// TIA Portal V20 export
DATA_BLOCK "InstCallEquipment"   // DB130
{ DB_Accessible_From_OPC_UA := 'FALSE' }
AUTHOR : ERsystem_FA2_DH. Kim
// stored: AssignedProDiagFB Unit1.Em6.ProDiag, DBAccessibleFromOPCUA false, DBAccessibleFromWebserver false, InstanceOfName Unit1.Em6.CallEquipment, InstanceOfType FB, Namespace Unit1.Em6
"Unit1.Em6.CallEquipment"
   // VAR_INPUT
   //    ZoneOperationEnable { ExternalWritable := 'False'} : "LWONIK_typeSafetyZoneManualOperation";
   // END_VAR
   // VAR_IN_OUT
   //    unitStatus : "LAF_typeUnitStatus";
   //    unitAlarmDB : "LAF_typeAlarms";
   //    emFeedback : "LUC_typeEmFeedback";
   // END_VAR
   // VAR
   //    InstSequenceStackTable { S7_SetPoint := 'True'} : "Unit1.Em6.Sequence_1_StackTable";
   //    InstSequenceGaugeRnR { S7_SetPoint := 'True'} : "Unit1.Em6.Sequence_10_GaugeRnR";
   //    InstSequenceUtility { S7_SetPoint := 'True'} : "Unit1.Em6.Sequence_20_Utility";
   //    instStackTableHomeJob1 { S7_SetPoint := 'True'} : "LAF_SelectJob";
   //    instStackTableMotionAutoJob2 { S7_SetPoint := 'True'} : "LAF_SelectJob";
   //    instStackTableRollerMoveJob12 { S7_SetPoint := 'True'} : "LAF_SelectJob";
   //    instStackTableRollerMoveJob13 { S7_SetPoint := 'True'} : "LAF_SelectJob";
   //    instStackTableSepaCleanJob14 { S7_SetPoint := 'True'} : "LAF_SelectJob";
   //    instStackTableAnodeMendrelJob22 { S7_SetPoint := 'True'} : "LAF_SelectJob";
   //    instStackTableCathodeMendrelJob23 { S7_SetPoint := 'True'} : "LAF_SelectJob";
   //    instStackTableVisionJob30 { S7_SetPoint := 'True'} : "LAF_SelectJob";
   //    instStackTableDownJob31 { S7_SetPoint := 'True'} : "LAF_SelectJob";
   //    instStackTableUnloadJob4 { S7_SetPoint := 'True'} : "LAF_SelectJob";
   //    instGaugeRnRReadyJob1 { S7_SetPoint := 'True'} : "LAF_SelectJob";
   //    instGaugeRnRVaccumJob2 { S7_SetPoint := 'True'} : "LAF_SelectJob";
   //    instGaugeRnRVisionJob3 { S7_SetPoint := 'True'} : "LAF_SelectJob";
   //    instGaugeRnRBlowJob4 { S7_SetPoint := 'True'} : "LAF_SelectJob";
   //    instUtilityFinalRollerHomeJob1 { S7_SetPoint := 'True'} : "LAF_SelectJob";
   //    instUtilityStackTableOutHomeJob2 { S7_SetPoint := 'True'} : "LAF_SelectJob";
   //    instUtilityAllMendrelOpenJob3 { S7_SetPoint := 'True'} : "LAF_SelectJob";
   //    instUtilityAllMendrelCloseJob4 { S7_SetPoint := 'True'} : "LAF_SelectJob";
   //    instCmStackTableElectrodeDetectSensor { S7_SetPoint := 'True'} : "LBC_DigitalSignalCn";
   //    instCmMasterVirtualAxisX : "LBC_Axis64Pos_TecPlcCn";
   //    instCmFinalRollerFrontAxisX : "LBC_Axis64Pos_TecPlcCn";
   //    instCmFinalRollerRearAxisX { S7_SetPoint := 'True'} : "LBC_Axis64Pos_TecPlcCn";
   //    instCmMendrelAnodeFrontAxisY { S7_SetPoint := 'True'} : "LBC_Axis64Pos_TecPlcCn";
   //    instCmMendrelAnodeFrontAxisZ { S7_SetPoint := 'True'} : "LBC_Axis64Pos_TecPlcCn";
   //    instCmMendrelAnodeRearAxisY { S7_SetPoint := 'True'} : "LBC_Axis64Pos_TecPlcCn";
   //    instCmMendrelAnodeRearAxisZ { S7_SetPoint := 'True'} : "LBC_Axis64Pos_TecPlcCn";
   //    instCmMendrelCathodeFrontAxisY { S7_SetPoint := 'True'} : "LBC_Axis64Pos_TecPlcCn";
   //    instCmMendrelCathodeFrontAxisZ { S7_SetPoint := 'True'} : "LBC_Axis64Pos_TecPlcCn";
   //    instCmMendrelCathodeRearAxisY { S7_SetPoint := 'True'} : "LBC_Axis64Pos_TecPlcCn";
   //    instCmMendrelCathodeRearAxisZ { S7_SetPoint := 'True'} : "LBC_Axis64Pos_TecPlcCn";
   //    instCmStackTableAxisZ { ExternalAccessible := 'False'; ExternalVisible := 'False'; ExternalWritable := 'False'; S7_SetPoint := 'True'} : "LBC_Axis64Pos_TecPlcCn";
   //    instCmStackTableOutFrontAxisZ { ExternalAccessible := 'False'; ExternalVisible := 'False'; ExternalWritable := 'False'; S7_SetPoint := 'True'} : "LBC_Axis64Pos_TecPlcCn";
   //    instCmStackTableOutRearAxisZ { ExternalAccessible := 'False'; ExternalVisible := 'False'; ExternalWritable := 'False'; S7_SetPoint := 'True'} : "LBC_Axis64Pos_TecPlcCn";
   //    instInterlockFinalRollerFrontAxisX : "LER_Axis64Pos_InterlockSummary";
   //    instInterlockFinalRollerRearAxisX : "LER_Axis64Pos_InterlockSummary";
   //    instInterlockMendrelAnodeFrontAxisY : "LER_Axis64Pos_InterlockSummary";
   //    instInterlockMendrelAnodeFrontAxisZ : "LER_Axis64Pos_InterlockSummary";
   //    instInterlockMendrelAnodeRearAxisY : "LER_Axis64Pos_InterlockSummary";
   //    instInterlockMendrelAnodeRearAxisZ : "LER_Axis64Pos_InterlockSummary";
   //    instInterlockMendrelCathodeFrontAxisY : "LER_Axis64Pos_InterlockSummary";
   //    instInterlockMendrelCathodeFrontAxisZ : "LER_Axis64Pos_InterlockSummary";
   //    instInterlockMendrelCathodeRearAxisY : "LER_Axis64Pos_InterlockSummary";
   //    instInterlockMendrelCathodeRearAxisZ : "LER_Axis64Pos_InterlockSummary";
   //    instInterlockStackTableAxisZ : "LER_Axis64Pos_InterlockSummary";
   //    instInterlockStackTableOutFrontAxisZ : "LER_Axis64Pos_InterlockSummary";
   //    instInterlockStackTableOutRearAxisZ : "LER_Axis64Pos_InterlockSummary";
   //    instFinalRollerFrontAxisXMCGearIn { S7_SetPoint := 'True'} : MC_GEARIN;
   //    instFinalRollerRearAxisXMCGearIn { S7_SetPoint := 'True'} : MC_GEARIN;
   //    instStackTableOutFrontAxisZMCGearIn { S7_SetPoint := 'True'} : MC_GEARIN;
   //    instStackTableOutRearAxisZMCGearIn { S7_SetPoint := 'True'} : MC_GEARIN;
   //    instFinalRollerFrontAxisXMCWirteParameter { S7_SetPoint := 'True'} : MC_WRITEPARAMETER;
   //    instFinalRollerRearAxisXMCWirteParameter { S7_SetPoint := 'True'} : MC_WRITEPARAMETER;
   //    instStackTableOutFrontAxisZMCWirteParameter { S7_SetPoint := 'True'} : MC_WRITEPARAMETER;
   //    instStackTableOutRearAxisZMCWirteParameter { S7_SetPoint := 'True'} : MC_WRITEPARAMETER;
   //    instCmMendrelCathodeFrontClamp { ExternalAccessible := 'False'; ExternalVisible := 'False'; ExternalWritable := 'False'; S7_SetPoint := 'True'} : "LBC_TwoWayActuatorCn";
   //    instCmMendrelAnodeFrontClamp { ExternalAccessible := 'False'; ExternalVisible := 'False'; ExternalWritable := 'False'; S7_SetPoint := 'True'} : "LBC_TwoWayActuatorCn";
   //    instCmMendrelCathodeRearClamp { ExternalAccessible := 'False'; ExternalVisible := 'False'; ExternalWritable := 'False'; S7_SetPoint := 'True'} : "LBC_TwoWayActuatorCn";
   //    instCmMendrelAnodeRearClamp { ExternalAccessible := 'False'; ExternalVisible := 'False'; ExternalWritable := 'False'; S7_SetPoint := 'True'} : "LBC_TwoWayActuatorCn";
   //    instcmStackTableVaccum { ExternalAccessible := 'False'; ExternalVisible := 'False'; ExternalWritable := 'False'; S7_SetPoint := 'True'} : "LBC_TwoWayActuatorCn";
   //    instcmStackTableGapPadUpDown { ExternalAccessible := 'False'; ExternalVisible := 'False'; ExternalWritable := 'False'; S7_SetPoint := 'True'} : "LBC_TwoWayActuatorCn";
   //    instCmStackTableVisionControllerInterface : "LER_Vision_XGX2000";
   //    instGapVisionConversion : "LER_StackTableVisionConversion";
   //    instManageAlarms { ExternalWritable := 'False'} : "LAF_ManageAlarms";
   //    instEventsPFE : "Unit1.Em6.EventsPFE";
   //    instLER_BrakeTestMendrelAnodeFrontAxisZ : "LER_BrakeTest";
   //    instLER_BrakeTestMendrelAnodeRearAxisZ { S7_SetPoint := 'True'} : "LER_BrakeTest";
   //    instLER_BrakeTestMendrelCathodeFrontAxisZ { S7_SetPoint := 'True'} : "LER_BrakeTest";
   //    instLER_BrakeTestMendrelCathodeRearAxisZ { S7_SetPoint := 'True'} : "LER_BrakeTest";
   //    instLER_BrakeTestStackTableAxisZ { S7_SetPoint := 'True'} : "LER_BrakeTest";
   //    instLER_BrakeTestStackTableOutFrontAxisZ { S7_SetPoint := 'True'} : "LER_BrakeTest";
   //    instLER_BrakeTestStackTableOutRearAxisZ { S7_SetPoint := 'True'} : "LER_BrakeTest";
   //    statUnitStatus { ExternalWritable := 'False'} : "LAF_typeUnitStatus";
   //    statSlmStatus : Struct
   //       running { ExternalWritable := 'False'} : Bool;
   //       powerOff { ExternalWritable := 'False'} : Bool;
   //    END_STRUCT;
   //    statAllBrakeTest { ExternalWritable := 'False'} : "LER_typeBrakeTestUnitCommands";
   //    statTonTime { ExternalAccessible := 'False'; ExternalVisible := 'False'; ExternalWritable := 'False'} : Array[0..1999] of TON_TIME;
   //    statTofTime { ExternalAccessible := 'False'; ExternalVisible := 'False'; ExternalWritable := 'False'} : Array[0..99] of TOF_TIME;
   //    statLReal { ExternalAccessible := 'False'; ExternalVisible := 'False'; ExternalWritable := 'False'} : Array[0..99] of LReal;
   //    statPulse { ExternalAccessible := 'False'; ExternalVisible := 'False'; ExternalWritable := 'False'} : Struct
   //       miscellaneous : Array[0..99] of Bool;
   //       workingDone : Array[0..99] of Bool;
   //       axisEnable : Array[0..99] of Bool;
   //       brakeTest : Array[0..99] of Bool;
   //    END_STRUCT;
   //    statEnableManualCmds : Bool := TRUE;
   //    scan_on : Bool;
   //    "*** Interlock Axis ***" { ExternalAccessible := 'False'; ExternalVisible := 'False'; ExternalWritable := 'False'} : Bool;
   //    instFinalRollerFrontAxisX_CW { S7_SetPoint := 'True'} : "Jog.LER_Axis";
   //    instFinalRollerFrontAxisX_CCW { S7_SetPoint := 'True'} : "Jog.LER_Axis";
   //    instFinalRollerFrontAxisX_Home { S7_SetPoint := 'True'} : "Homing.LER_Axis";
   //    instFinalRollerFrontAxisX_Position { S7_SetPoint := 'True'} : Array[0..6] of "Position.LER_Axis";
   //    instFinalRollerRearAxisX_CW { S7_SetPoint := 'True'} : "Jog.LER_Axis";
   //    instFinalRollerRearAxisX_CCW { S7_SetPoint := 'True'} : "Jog.LER_Axis";
   //    instFinalRollerRearAxisX_Home { S7_SetPoint := 'True'} : "Homing.LER_Axis";
   //    instFinalRollerRearAxisX_Position { S7_SetPoint := 'True'} : Array[0..6] of "Position.LER_Axis";
   //    instMendrelAnodeFrontAxisY_CW { S7_SetPoint := 'True'} : "Jog.LER_Axis";
   //    instMendrelAnodeFrontAxisY_CCW { S7_SetPoint := 'True'} : "Jog.LER_Axis";
   //    instMendrelAnodeFrontAxisY_Home { S7_SetPoint := 'True'} : "Homing.LER_Axis";
   //    instMendrelAnodeFrontAxisY_Position { S7_SetPoint := 'True'} : Array[0..15] of "Position.LER_Axis";
   //    instMendrelAnodeFrontAxisZ_CW { S7_SetPoint := 'True'} : "Jog.LER_Axis";
   //    instMendrelAnodeFrontAxisZ_CCW { S7_SetPoint := 'True'} : "Jog.LER_Axis";
   //    instMendrelAnodeFrontAxisZ_Home { S7_SetPoint := 'True'} : "Homing.LER_Axis";
   //    instMendrelAnodeFrontAxisZ_Position { S7_SetPoint := 'True'} : Array[0..6] of "Position.LER_Axis";
   //    instMendrelAnodeRearAxisY_CW { S7_SetPoint := 'True'} : "Jog.LER_Axis";
   //    instMendrelAnodeRearAxisY_CCW { S7_SetPoint := 'True'} : "Jog.LER_Axis";
   //    instMendrelAnodeRearAxisY_Home { S7_SetPoint := 'True'} : "Homing.LER_Axis";
   //    instMendrelAnodeRearAxisY_Position { S7_SetPoint := 'True'} : Array[0..6] of "Position.LER_Axis";
   //    instMendrelAnodeRearAxisZ_CW { S7_SetPoint := 'True'} : "Jog.LER_Axis";
   //    instMendrelAnodeRearAxisZ_CCW { S7_SetPoint := 'True'} : "Jog.LER_Axis";
   //    instMendrelAnodeRearAxisZ_Home { S7_SetPoint := 'True'} : "Homing.LER_Axis";
   //    instMendrelAnodeRearAxisZ_Position { S7_SetPoint := 'True'} : Array[0..6] of "Position.LER_Axis";
   //    instMendrelCathodeFrontAxisY_CW { S7_SetPoint := 'True'} : "Jog.LER_Axis";
   //    instMendrelCathodeFrontAxisY_CCW { S7_SetPoint := 'True'} : "Jog.LER_Axis";
   //    instMendrelCathodeFrontAxisY_Home { S7_SetPoint := 'True'} : "Homing.LER_Axis";
   //    instMendrelCathodeFrontAxisY_Position { S7_SetPoint := 'True'} : Array[0..6] of "Position.LER_Axis";
   //    instMendrelCathodeFrontAxisZ_CW { S7_SetPoint := 'True'} : "Jog.LER_Axis";
   //    instMendrelCathodeFrontAxisZ_CCW { S7_SetPoint := 'True'} : "Jog.LER_Axis";
   //    instMendrelCathodeFrontAxisZ_Home { S7_SetPoint := 'True'} : "Homing.LER_Axis";
   //    instMendrelCathodeFrontAxisZ_Position { S7_SetPoint := 'True'} : Array[0..6] of "Position.LER_Axis";
   //    instMendrelCathodeRearAxisY_CW { S7_SetPoint := 'True'} : "Jog.LER_Axis";
   //    instMendrelCathodeRearAxisY_CCW { S7_SetPoint := 'True'} : "Jog.LER_Axis";
   //    instMendrelCathodeRearAxisY_Home { S7_SetPoint := 'True'} : "Homing.LER_Axis";
   //    instMendrelCathodeRearAxisY_Position { S7_SetPoint := 'True'} : Array[0..6] of "Position.LER_Axis";
   //    instMendrelCathodeRearAxisZ_CW { S7_SetPoint := 'True'} : "Jog.LER_Axis";
   //    instMendrelCathodeRearAxisZ_CCW { S7_SetPoint := 'True'} : "Jog.LER_Axis";
   //    instMendrelCathodeRearAxisZ_Home { S7_SetPoint := 'True'} : "Homing.LER_Axis";
   //    instMendrelCathodeRearAxisZ_Position { S7_SetPoint := 'True'} : Array[0..6] of "Position.LER_Axis";
   //    instStackTableAxisZ_CW { S7_SetPoint := 'True'} : "Jog.LER_Axis";
   //    instStackTableAxisZ_CCW { S7_SetPoint := 'True'} : "Jog.LER_Axis";
   //    instStackTableAxisZ_Home { S7_SetPoint := 'True'} : "Homing.LER_Axis";
   //    instStackTableAxisZ_Position { S7_SetPoint := 'True'} : Array[0..6] of "Position.LER_Axis";
   //    instStackTableOutFrontAxisZ_CW { S7_SetPoint := 'True'} : "Jog.LER_Axis";
   //    instStackTableOutFrontAxisZ_CCW { S7_SetPoint := 'True'} : "Jog.LER_Axis";
   //    instStackTableOutFrontAxisZ_Home { S7_SetPoint := 'True'} : "Homing.LER_Axis";
   //    instStackTableOutFrontAxisZ_Position { S7_SetPoint := 'True'} : Array[0..6] of "Position.LER_Axis";
   //    instStackTableOutRearAxisZ_CW { S7_SetPoint := 'True'} : "Jog.LER_Axis";
   //    instStackTableOutRearAxisZ_CCW { S7_SetPoint := 'True'} : "Jog.LER_Axis";
   //    instStackTableOutRearAxisZ_Home { S7_SetPoint := 'True'} : "Homing.LER_Axis";
   //    instStackTableOutRearAxisZ_Position { S7_SetPoint := 'True'} : Array[0..6] of "Position.LER_Axis";
   //    "*** Interlock Actuator ******" { ExternalAccessible := 'False'; ExternalVisible := 'False'; ExternalWritable := 'False'} : Bool;
   //    instCmMendrelCathodeFrontClampInterlock : Array[0..1] of "Cylinder.LER_Actuator";
   //    instCmMendrelAnodeFrontClampInterlock { S7_SetPoint := 'True'} : Array[0..1] of "Cylinder.LER_Actuator";
   //    instCmMendrelCathodeRearClampInterlock { S7_SetPoint := 'True'} : Array[0..1] of "Cylinder.LER_Actuator";
   //    instCmMendrelAnodeRearClampInterlock { S7_SetPoint := 'True'} : Array[0..1] of "Cylinder.LER_Actuator";
   //    instcmStackTableVaccumInterlock { S7_SetPoint := 'True'} : Array[0..1] of "Cylinder.LER_Actuator";
   //    instcmStackTableGapPadUpDownInterlock { S7_SetPoint := 'True'} : Array[0..1] of "Cylinder.LER_Actuator";
   //    AXIS21 : "LER_CM_Name";
   //    AXIS26 : "LER_CM_Name";
   //    AXIS31 : "LER_CM_Name";
   //    Cylinder33 : "LER_CM_Name";
   //    Vaccum20 : "LER_CM_Name";
   //    instFinalRollerGearInVel : MC_GEARINVELOCITY;
   //    instStackTableOutGearInVel : MC_GEARINVELOCITY;
   //    instFinalRollerGantryHoming : "LER_GantryHoming";
   //    instStackTableOutGantryHoming : "LER_GantryHoming";
   //    citi_Ptrig : Array[0..20] of Bool;
   //    citiTon : Array[0..20] of TON_TIME;
   //    citi : Time;
   //    citiTest : Array[0..20] of Bool;
   // END_VAR
BEGIN
   ZoneOperationEnable.autoStartEnable := FALSE;
   ZoneOperationEnable.doorLockEnable := TRUE;
   ZoneOperationEnable.doorUnlockEnable := TRUE;
   ZoneOperationEnable.rc_AutoEnable := FALSE;
   ZoneOperationEnable.rc_RollChangeEnable := FALSE;
   ZoneOperationEnable.rc_DoorLockEnable := TRUE;
   ZoneOperationEnable.rc_DoorUnlockEnable := TRUE;
   ZoneOperationEnable.hmiOperationEnable := TRUE;
   ZoneOperationEnable.phmiOperationEnable := FALSE;
   instCmStackTableElectrodeDetectSensor.enable := TRUE;
   instCmStackTableElectrodeDetectSensor.parentReferenceDesignator := WSTRING#'';
   instCmStackTableElectrodeDetectSensor.digitalValue := FALSE;
   instCmStackTableElectrodeDetectSensor.simulatedDigitalValue := FALSE;
   instCmStackTableElectrodeDetectSensor.statProcessValues.enable := TRUE;
   instCmStackTableElectrodeDetectSensor.statProcessValues.referenceDesignator := WSTRING#'DigitalSignal';
   instCmStackTableElectrodeDetectSensor.statProcessValues.simulation := FALSE;
   instCmStackTableElectrodeDetectSensor.statProcessValues.processValue := FALSE;
   instCmStackTableElectrodeDetectSensor.statProcessValues.error := FALSE;
   instCmStackTableElectrodeDetectSensor.statProcessValues.status := 16#0000;
   instCmStackTableElectrodeDetectSensor.statDiagnostics.status := 16#0000;
   instCmStackTableElectrodeDetectSensor.statDiagnostics.subfunctionStatus := 16#0000;
   instCmStackTableElectrodeDetectSensor.statDiagnostics.stateNumber := 0;
   instCmStackTableElectrodeDetectSensor.statEmptyDiagnostics.status := 16#0000;
   instCmStackTableElectrodeDetectSensor.statEmptyDiagnostics.subfunctionStatus := 16#0000;
   instCmStackTableElectrodeDetectSensor.statEmptyDiagnostics.stateNumber := 0;
   instCmStackTableElectrodeDetectSensor.instOnDelay.PT := T#0MS;
   instCmStackTableElectrodeDetectSensor.instOnDelay.IN := FALSE;
   instCmStackTableElectrodeDetectSensor.instOffDelay.PT := T#0MS;
   instCmStackTableElectrodeDetectSensor.instOffDelay.IN := FALSE;
   instCmStackTableElectrodeDetectSensor.statDisableAlarms := FALSE;
   instCmStackTableElectrodeDetectSensor.statErrorState := 16#0000;
   instCmStackTableElectrodeDetectSensor.statFirstCall := FALSE;
   instCmStackTableElectrodeDetectSensor.statResetPrevious := FALSE;
   instCmStackTableElectrodeDetectSensor.statEnablePrevious := TRUE;
   instCmStackTableElectrodeDetectSensor.statProcessValuePrevious := FALSE;
   instCmMendrelCathodeFrontClamp.enable := TRUE;
   instCmMendrelCathodeFrontClamp.parentReferenceDesignator := WSTRING#'';
   instCmMendrelCathodeFrontClamp.feedbackHomePos := FALSE;
   instCmMendrelCathodeFrontClamp.feedbackWorkPos := FALSE;
   instCmMendrelCathodeFrontClamp.enableManualCmds := TRUE;
   instCmMendrelCathodeFrontClamp.interlockWorkPos := TRUE;
   instCmMendrelCathodeFrontClamp.interlockHomePos := TRUE;
   instCmMendrelCathodeFrontClamp.goToHomePos := FALSE;
   instCmMendrelCathodeFrontClamp.goToWorkPos := FALSE;
   instCmMendrelCathodeFrontClamp.statProcessValues.enable := TRUE;
   instCmMendrelCathodeFrontClamp.statProcessValues.referenceDesignator := WSTRING#'MendrelCathodeFrontClamp';
   instCmMendrelCathodeFrontClamp.statProcessValues.commandHomePos := FALSE;
   instCmMendrelCathodeFrontClamp.statProcessValues.commandWorkPos := FALSE;
   instCmMendrelCathodeFrontClamp.statProcessValues.goToHomePos := FALSE;
   instCmMendrelCathodeFrontClamp.statProcessValues.goToWorkPos := FALSE;
   instCmMendrelCathodeFrontClamp.statProcessValues.inHomePos := FALSE;
   instCmMendrelCathodeFrontClamp.statProcessValues.inWorkPos := FALSE;
   instCmMendrelCathodeFrontClamp.statProcessValues.reset := FALSE;
   instCmMendrelCathodeFrontClamp.statProcessValues.enableManualCmds := TRUE;
   instCmMendrelCathodeFrontClamp.statProcessValues.error := FALSE;
   instCmMendrelCathodeFrontClamp.statProcessValues.interlockHomePos := TRUE;
   instCmMendrelCathodeFrontClamp.statProcessValues.interlockWorkPos := TRUE;
   instCmMendrelCathodeFrontClamp.statProcessValues.status := 16#7003;
   instCmMendrelCathodeFrontClamp.statProcessValues.interlockWarningWorkPos := FALSE;
   instCmMendrelCathodeFrontClamp.statProcessValues.interlockWarningHomePos := FALSE;
   instCmMendrelCathodeFrontClamp.statCurrentInputs.commandHomePos := FALSE;
   instCmMendrelCathodeFrontClamp.statCurrentInputs.commandWorkPos := FALSE;
   instCmMendrelCathodeFrontClamp.statCurrentInputs.reset := FALSE;
   instCmMendrelCathodeFrontClamp.statPreviousInputs.commandHomePos := FALSE;
   instCmMendrelCathodeFrontClamp.statPreviousInputs.commandWorkPos := FALSE;
   instCmMendrelCathodeFrontClamp.statPreviousInputs.reset := FALSE;
   instCmMendrelCathodeFrontClamp.statCurrentInterface.commandHomePos := FALSE;
   instCmMendrelCathodeFrontClamp.statCurrentInterface.commandWorkPos := FALSE;
   instCmMendrelCathodeFrontClamp.statCurrentInterface.reset := FALSE;
   instCmMendrelCathodeFrontClamp.statPreviousInterface.commandHomePos := FALSE;
   instCmMendrelCathodeFrontClamp.statPreviousInterface.commandWorkPos := FALSE;
   instCmMendrelCathodeFrontClamp.statPreviousInterface.reset := FALSE;
   instCmMendrelCathodeFrontClamp.statEmptyDiagnostics.status := 16#0000;
   instCmMendrelCathodeFrontClamp.statEmptyDiagnostics.subfunctionStatus := 16#0000;
   instCmMendrelCathodeFrontClamp.statEmptyDiagnostics.stateNumber := 0;
   instCmMendrelCathodeFrontClamp.instTimerReachPos.PT := T#0MS;
   instCmMendrelCathodeFrontClamp.instTimerReachPos.IN := FALSE;
   instCmMendrelCathodeFrontClamp.instTimerLeavePos.PT := T#0MS;
   instCmMendrelCathodeFrontClamp.instTimerLeavePos.IN := FALSE;
   instCmMendrelCathodeFrontClamp.instTimerDiscrepancyCheck.PT := T#0MS;
   instCmMendrelCathodeFrontClamp.instTimerDiscrepancyCheck.IN := FALSE;
   instCmMendrelCathodeFrontClamp.statDisableAlarms := FALSE;
   instCmMendrelCathodeFrontClamp.statDiagnostics.status := 16#7003;
   instCmMendrelCathodeFrontClamp.statDiagnostics.subfunctionStatus := 16#0000;
   instCmMendrelCathodeFrontClamp.statDiagnostics.stateNumber := 0;
   instCmMendrelCathodeFrontClamp.statEnablePrevious := TRUE;
   instCmMendrelCathodeFrontClamp.statFirstCall := FALSE;
   instCmMendrelCathodeFrontClamp.statResetPrevious := FALSE;
   instCmMendrelCathodeFrontClamp.statValid := TRUE;
   instCmMendrelCathodeFrontClamp.statBusy := TRUE;
   instCmMendrelCathodeFrontClamp.statError := FALSE;
   instCmMendrelCathodeFrontClamp.statInterlockWorkOff := FALSE;
   instCmMendrelCathodeFrontClamp.statInterlockHomeOff := FALSE;
   instCmMendrelCathodeFrontClamp.statFbState := 50;
   instCmMendrelCathodeFrontClamp.statFbStatePrevious := 50;
   instCmMendrelCathodeFrontClamp.statErrorUserCleared := FALSE;
   instCmMendrelCathodeFrontClamp.statErrorAutoCleared := FALSE;
   instCmMendrelCathodeFrontClamp.statErrorState := 16#0000;
   instCmMendrelCathodeFrontClamp.statDisablingCompleted := FALSE;
   instCmMendrelCathodeFrontClamp.statFeedbackHomePos := FALSE;
   instCmMendrelCathodeFrontClamp.statFeedbackWorkPos := FALSE;
   instCmMendrelAnodeFrontClamp.enable := TRUE;
   instCmMendrelAnodeFrontClamp.parentReferenceDesignator := WSTRING#'';
   instCmMendrelAnodeFrontClamp.feedbackHomePos := FALSE;
   instCmMendrelAnodeFrontClamp.feedbackWorkPos := FALSE;
   instCmMendrelAnodeFrontClamp.enableManualCmds := TRUE;
   instCmMendrelAnodeFrontClamp.interlockWorkPos := TRUE;
   instCmMendrelAnodeFrontClamp.interlockHomePos := TRUE;
   instCmMendrelAnodeFrontClamp.goToHomePos := FALSE;
   instCmMendrelAnodeFrontClamp.goToWorkPos := FALSE;
   instCmMendrelAnodeFrontClamp.statProcessValues.enable := TRUE;
   instCmMendrelAnodeFrontClamp.statProcessValues.referenceDesignator := WSTRING#'MendrelAnodeFrontClamp';
   instCmMendrelAnodeFrontClamp.statProcessValues.commandHomePos := FALSE;
   instCmMendrelAnodeFrontClamp.statProcessValues.commandWorkPos := FALSE;
   instCmMendrelAnodeFrontClamp.statProcessValues.goToHomePos := FALSE;
   instCmMendrelAnodeFrontClamp.statProcessValues.goToWorkPos := FALSE;
   instCmMendrelAnodeFrontClamp.statProcessValues.inHomePos := FALSE;
   instCmMendrelAnodeFrontClamp.statProcessValues.inWorkPos := FALSE;
   instCmMendrelAnodeFrontClamp.statProcessValues.reset := FALSE;
   instCmMendrelAnodeFrontClamp.statProcessValues.enableManualCmds := TRUE;
   instCmMendrelAnodeFrontClamp.statProcessValues.error := FALSE;
   instCmMendrelAnodeFrontClamp.statProcessValues.interlockHomePos := TRUE;
   instCmMendrelAnodeFrontClamp.statProcessValues.interlockWorkPos := TRUE;
   instCmMendrelAnodeFrontClamp.statProcessValues.status := 16#7003;
   instCmMendrelAnodeFrontClamp.statProcessValues.interlockWarningWorkPos := FALSE;
   instCmMendrelAnodeFrontClamp.statProcessValues.interlockWarningHomePos := FALSE;
   instCmMendrelAnodeFrontClamp.statCurrentInputs.commandHomePos := FALSE;
   instCmMendrelAnodeFrontClamp.statCurrentInputs.commandWorkPos := FALSE;
   instCmMendrelAnodeFrontClamp.statCurrentInputs.reset := FALSE;
   instCmMendrelAnodeFrontClamp.statPreviousInputs.commandHomePos := FALSE;
   instCmMendrelAnodeFrontClamp.statPreviousInputs.commandWorkPos := FALSE;
   instCmMendrelAnodeFrontClamp.statPreviousInputs.reset := FALSE;
   instCmMendrelAnodeFrontClamp.statCurrentInterface.commandHomePos := FALSE;
   instCmMendrelAnodeFrontClamp.statCurrentInterface.commandWorkPos := FALSE;
   instCmMendrelAnodeFrontClamp.statCurrentInterface.reset := FALSE;
   instCmMendrelAnodeFrontClamp.statPreviousInterface.commandHomePos := FALSE;
   instCmMendrelAnodeFrontClamp.statPreviousInterface.commandWorkPos := FALSE;
   instCmMendrelAnodeFrontClamp.statPreviousInterface.reset := FALSE;
   instCmMendrelAnodeFrontClamp.statEmptyDiagnostics.status := 16#0000;
   instCmMendrelAnodeFrontClamp.statEmptyDiagnostics.subfunctionStatus := 16#0000;
   instCmMendrelAnodeFrontClamp.statEmptyDiagnostics.stateNumber := 0;
   instCmMendrelAnodeFrontClamp.instTimerReachPos.PT := T#0MS;
   instCmMendrelAnodeFrontClamp.instTimerReachPos.IN := FALSE;
   instCmMendrelAnodeFrontClamp.instTimerLeavePos.PT := T#0MS;
   instCmMendrelAnodeFrontClamp.instTimerLeavePos.IN := FALSE;
   instCmMendrelAnodeFrontClamp.instTimerDiscrepancyCheck.PT := T#0MS;
   instCmMendrelAnodeFrontClamp.instTimerDiscrepancyCheck.IN := FALSE;
   instCmMendrelAnodeFrontClamp.statDisableAlarms := FALSE;
   instCmMendrelAnodeFrontClamp.statDiagnostics.status := 16#7003;
   instCmMendrelAnodeFrontClamp.statDiagnostics.subfunctionStatus := 16#0000;
   instCmMendrelAnodeFrontClamp.statDiagnostics.stateNumber := 0;
   instCmMendrelAnodeFrontClamp.statEnablePrevious := TRUE;
   instCmMendrelAnodeFrontClamp.statFirstCall := FALSE;
   instCmMendrelAnodeFrontClamp.statResetPrevious := FALSE;
   instCmMendrelAnodeFrontClamp.statValid := TRUE;
   instCmMendrelAnodeFrontClamp.statBusy := TRUE;
   instCmMendrelAnodeFrontClamp.statError := FALSE;
   instCmMendrelAnodeFrontClamp.statInterlockWorkOff := FALSE;
   instCmMendrelAnodeFrontClamp.statInterlockHomeOff := FALSE;
   instCmMendrelAnodeFrontClamp.statFbState := 50;
   instCmMendrelAnodeFrontClamp.statFbStatePrevious := 50;
   instCmMendrelAnodeFrontClamp.statErrorUserCleared := FALSE;
   instCmMendrelAnodeFrontClamp.statErrorAutoCleared := FALSE;
   instCmMendrelAnodeFrontClamp.statErrorState := 16#0000;
   instCmMendrelAnodeFrontClamp.statDisablingCompleted := FALSE;
   instCmMendrelAnodeFrontClamp.statFeedbackHomePos := FALSE;
   instCmMendrelAnodeFrontClamp.statFeedbackWorkPos := FALSE;
   instCmMendrelCathodeRearClamp.enable := TRUE;
   instCmMendrelCathodeRearClamp.parentReferenceDesignator := WSTRING#'';
   instCmMendrelCathodeRearClamp.feedbackHomePos := FALSE;
   instCmMendrelCathodeRearClamp.feedbackWorkPos := FALSE;
   instCmMendrelCathodeRearClamp.enableManualCmds := TRUE;
   instCmMendrelCathodeRearClamp.interlockWorkPos := TRUE;
   instCmMendrelCathodeRearClamp.interlockHomePos := TRUE;
   instCmMendrelCathodeRearClamp.goToHomePos := FALSE;
   instCmMendrelCathodeRearClamp.goToWorkPos := FALSE;
   instCmMendrelCathodeRearClamp.statProcessValues.enable := TRUE;
   instCmMendrelCathodeRearClamp.statProcessValues.referenceDesignator := WSTRING#'MendrelCathodeRearClamp';
   instCmMendrelCathodeRearClamp.statProcessValues.commandHomePos := FALSE;
   instCmMendrelCathodeRearClamp.statProcessValues.commandWorkPos := FALSE;
   instCmMendrelCathodeRearClamp.statProcessValues.goToHomePos := FALSE;
   instCmMendrelCathodeRearClamp.statProcessValues.goToWorkPos := FALSE;
   instCmMendrelCathodeRearClamp.statProcessValues.inHomePos := FALSE;
   instCmMendrelCathodeRearClamp.statProcessValues.inWorkPos := FALSE;
   instCmMendrelCathodeRearClamp.statProcessValues.reset := FALSE;
   instCmMendrelCathodeRearClamp.statProcessValues.enableManualCmds := TRUE;
   instCmMendrelCathodeRearClamp.statProcessValues.error := FALSE;
   instCmMendrelCathodeRearClamp.statProcessValues.interlockHomePos := TRUE;
   instCmMendrelCathodeRearClamp.statProcessValues.interlockWorkPos := TRUE;
   instCmMendrelCathodeRearClamp.statProcessValues.status := 16#7003;
   instCmMendrelCathodeRearClamp.statProcessValues.interlockWarningWorkPos := FALSE;
   instCmMendrelCathodeRearClamp.statProcessValues.interlockWarningHomePos := FALSE;
   instCmMendrelCathodeRearClamp.statCurrentInputs.commandHomePos := FALSE;
   instCmMendrelCathodeRearClamp.statCurrentInputs.commandWorkPos := FALSE;
   instCmMendrelCathodeRearClamp.statCurrentInputs.reset := FALSE;
   instCmMendrelCathodeRearClamp.statPreviousInputs.commandHomePos := FALSE;
   instCmMendrelCathodeRearClamp.statPreviousInputs.commandWorkPos := FALSE;
   instCmMendrelCathodeRearClamp.statPreviousInputs.reset := FALSE;
   instCmMendrelCathodeRearClamp.statCurrentInterface.commandHomePos := FALSE;
   instCmMendrelCathodeRearClamp.statCurrentInterface.commandWorkPos := FALSE;
   instCmMendrelCathodeRearClamp.statCurrentInterface.reset := FALSE;
   instCmMendrelCathodeRearClamp.statPreviousInterface.commandHomePos := FALSE;
   instCmMendrelCathodeRearClamp.statPreviousInterface.commandWorkPos := FALSE;
   instCmMendrelCathodeRearClamp.statPreviousInterface.reset := FALSE;
   instCmMendrelCathodeRearClamp.statEmptyDiagnostics.status := 16#0000;
   instCmMendrelCathodeRearClamp.statEmptyDiagnostics.subfunctionStatus := 16#0000;
   instCmMendrelCathodeRearClamp.statEmptyDiagnostics.stateNumber := 0;
   instCmMendrelCathodeRearClamp.instTimerReachPos.PT := T#0MS;
   instCmMendrelCathodeRearClamp.instTimerReachPos.IN := FALSE;
   instCmMendrelCathodeRearClamp.instTimerLeavePos.PT := T#0MS;
   instCmMendrelCathodeRearClamp.instTimerLeavePos.IN := FALSE;
   instCmMendrelCathodeRearClamp.instTimerDiscrepancyCheck.PT := T#0MS;
   instCmMendrelCathodeRearClamp.instTimerDiscrepancyCheck.IN := FALSE;
   instCmMendrelCathodeRearClamp.statDisableAlarms := FALSE;
   instCmMendrelCathodeRearClamp.statDiagnostics.status := 16#7003;
   instCmMendrelCathodeRearClamp.statDiagnostics.subfunctionStatus := 16#0000;
   instCmMendrelCathodeRearClamp.statDiagnostics.stateNumber := 0;
   instCmMendrelCathodeRearClamp.statEnablePrevious := TRUE;
   instCmMendrelCathodeRearClamp.statFirstCall := FALSE;
   instCmMendrelCathodeRearClamp.statResetPrevious := FALSE;
   instCmMendrelCathodeRearClamp.statValid := TRUE;
   instCmMendrelCathodeRearClamp.statBusy := TRUE;
   instCmMendrelCathodeRearClamp.statError := FALSE;
   instCmMendrelCathodeRearClamp.statInterlockWorkOff := FALSE;
   instCmMendrelCathodeRearClamp.statInterlockHomeOff := FALSE;
   instCmMendrelCathodeRearClamp.statFbState := 50;
   instCmMendrelCathodeRearClamp.statFbStatePrevious := 50;
   instCmMendrelCathodeRearClamp.statErrorUserCleared := FALSE;
   instCmMendrelCathodeRearClamp.statErrorAutoCleared := FALSE;
   instCmMendrelCathodeRearClamp.statErrorState := 16#0000;
   instCmMendrelCathodeRearClamp.statDisablingCompleted := FALSE;
   instCmMendrelCathodeRearClamp.statFeedbackHomePos := FALSE;
   instCmMendrelCathodeRearClamp.statFeedbackWorkPos := FALSE;
   instCmMendrelAnodeRearClamp.enable := TRUE;
   instCmMendrelAnodeRearClamp.parentReferenceDesignator := WSTRING#'';
   instCmMendrelAnodeRearClamp.feedbackHomePos := FALSE;
   instCmMendrelAnodeRearClamp.feedbackWorkPos := FALSE;
   instCmMendrelAnodeRearClamp.enableManualCmds := TRUE;
   instCmMendrelAnodeRearClamp.interlockWorkPos := TRUE;
   instCmMendrelAnodeRearClamp.interlockHomePos := TRUE;
   instCmMendrelAnodeRearClamp.goToHomePos := FALSE;
   instCmMendrelAnodeRearClamp.goToWorkPos := FALSE;
   instCmMendrelAnodeRearClamp.statProcessValues.enable := TRUE;
   instCmMendrelAnodeRearClamp.statProcessValues.referenceDesignator := WSTRING#'MendrelAnodeRearClamp';
   instCmMendrelAnodeRearClamp.statProcessValues.commandHomePos := FALSE;
   instCmMendrelAnodeRearClamp.statProcessValues.commandWorkPos := FALSE;
   instCmMendrelAnodeRearClamp.statProcessValues.goToHomePos := FALSE;
   instCmMendrelAnodeRearClamp.statProcessValues.goToWorkPos := FALSE;
   instCmMendrelAnodeRearClamp.statProcessValues.inHomePos := FALSE;
   instCmMendrelAnodeRearClamp.statProcessValues.inWorkPos := FALSE;
   instCmMendrelAnodeRearClamp.statProcessValues.reset := FALSE;
   instCmMendrelAnodeRearClamp.statProcessValues.enableManualCmds := TRUE;
   instCmMendrelAnodeRearClamp.statProcessValues.error := FALSE;
   instCmMendrelAnodeRearClamp.statProcessValues.interlockHomePos := TRUE;
   instCmMendrelAnodeRearClamp.statProcessValues.interlockWorkPos := TRUE;
   instCmMendrelAnodeRearClamp.statProcessValues.status := 16#7003;
   instCmMendrelAnodeRearClamp.statProcessValues.interlockWarningWorkPos := FALSE;
   instCmMendrelAnodeRearClamp.statProcessValues.interlockWarningHomePos := FALSE;
   instCmMendrelAnodeRearClamp.statCurrentInputs.commandHomePos := FALSE;
   instCmMendrelAnodeRearClamp.statCurrentInputs.commandWorkPos := FALSE;
   instCmMendrelAnodeRearClamp.statCurrentInputs.reset := FALSE;
   instCmMendrelAnodeRearClamp.statPreviousInputs.commandHomePos := FALSE;
   instCmMendrelAnodeRearClamp.statPreviousInputs.commandWorkPos := FALSE;
   instCmMendrelAnodeRearClamp.statPreviousInputs.reset := FALSE;
   instCmMendrelAnodeRearClamp.statCurrentInterface.commandHomePos := FALSE;
   instCmMendrelAnodeRearClamp.statCurrentInterface.commandWorkPos := FALSE;
   instCmMendrelAnodeRearClamp.statCurrentInterface.reset := FALSE;
   instCmMendrelAnodeRearClamp.statPreviousInterface.commandHomePos := FALSE;
   instCmMendrelAnodeRearClamp.statPreviousInterface.commandWorkPos := FALSE;
   instCmMendrelAnodeRearClamp.statPreviousInterface.reset := FALSE;
   instCmMendrelAnodeRearClamp.statEmptyDiagnostics.status := 16#0000;
   instCmMendrelAnodeRearClamp.statEmptyDiagnostics.subfunctionStatus := 16#0000;
   instCmMendrelAnodeRearClamp.statEmptyDiagnostics.stateNumber := 0;
   instCmMendrelAnodeRearClamp.instTimerReachPos.PT := T#0MS;
   instCmMendrelAnodeRearClamp.instTimerReachPos.IN := FALSE;
   instCmMendrelAnodeRearClamp.instTimerLeavePos.PT := T#0MS;
   instCmMendrelAnodeRearClamp.instTimerLeavePos.IN := FALSE;
   instCmMendrelAnodeRearClamp.instTimerDiscrepancyCheck.PT := T#0MS;
   instCmMendrelAnodeRearClamp.instTimerDiscrepancyCheck.IN := FALSE;
   instCmMendrelAnodeRearClamp.statDisableAlarms := FALSE;
   instCmMendrelAnodeRearClamp.statDiagnostics.status := 16#7003;
   instCmMendrelAnodeRearClamp.statDiagnostics.subfunctionStatus := 16#0000;
   instCmMendrelAnodeRearClamp.statDiagnostics.stateNumber := 0;
   instCmMendrelAnodeRearClamp.statEnablePrevious := TRUE;
   instCmMendrelAnodeRearClamp.statFirstCall := FALSE;
   instCmMendrelAnodeRearClamp.statResetPrevious := FALSE;
   instCmMendrelAnodeRearClamp.statValid := TRUE;
   instCmMendrelAnodeRearClamp.statBusy := TRUE;
   instCmMendrelAnodeRearClamp.statError := FALSE;
   instCmMendrelAnodeRearClamp.statInterlockWorkOff := FALSE;
   instCmMendrelAnodeRearClamp.statInterlockHomeOff := FALSE;
   instCmMendrelAnodeRearClamp.statFbState := 50;
   instCmMendrelAnodeRearClamp.statFbStatePrevious := 50;
   instCmMendrelAnodeRearClamp.statErrorUserCleared := FALSE;
   instCmMendrelAnodeRearClamp.statErrorAutoCleared := FALSE;
   instCmMendrelAnodeRearClamp.statErrorState := 16#0000;
   instCmMendrelAnodeRearClamp.statDisablingCompleted := FALSE;
   instCmMendrelAnodeRearClamp.statFeedbackHomePos := FALSE;
   instCmMendrelAnodeRearClamp.statFeedbackWorkPos := FALSE;
   instcmStackTableVaccum.enable := TRUE;
   instcmStackTableVaccum.parentReferenceDesignator := WSTRING#'';
   instcmStackTableVaccum.feedbackHomePos := TRUE;
   instcmStackTableVaccum.feedbackWorkPos := FALSE;
   instcmStackTableVaccum.enableManualCmds := TRUE;
   instcmStackTableVaccum.interlockWorkPos := TRUE;
   instcmStackTableVaccum.interlockHomePos := TRUE;
   instcmStackTableVaccum.goToHomePos := FALSE;
   instcmStackTableVaccum.goToWorkPos := FALSE;
   instcmStackTableVaccum.statProcessValues.enable := TRUE;
   instcmStackTableVaccum.statProcessValues.referenceDesignator := WSTRING#'StackTableVaccum';
   instcmStackTableVaccum.statProcessValues.commandHomePos := FALSE;
   instcmStackTableVaccum.statProcessValues.commandWorkPos := FALSE;
   instcmStackTableVaccum.statProcessValues.goToHomePos := FALSE;
   instcmStackTableVaccum.statProcessValues.goToWorkPos := FALSE;
   instcmStackTableVaccum.statProcessValues.inHomePos := FALSE;
   instcmStackTableVaccum.statProcessValues.inWorkPos := FALSE;
   instcmStackTableVaccum.statProcessValues.reset := FALSE;
   instcmStackTableVaccum.statProcessValues.enableManualCmds := TRUE;
   instcmStackTableVaccum.statProcessValues.error := FALSE;
   instcmStackTableVaccum.statProcessValues.interlockHomePos := TRUE;
   instcmStackTableVaccum.statProcessValues.interlockWorkPos := TRUE;
   instcmStackTableVaccum.statProcessValues.status := 16#7003;
   instcmStackTableVaccum.statProcessValues.interlockWarningWorkPos := FALSE;
   instcmStackTableVaccum.statProcessValues.interlockWarningHomePos := FALSE;
   instcmStackTableVaccum.statCurrentInputs.commandHomePos := FALSE;
   instcmStackTableVaccum.statCurrentInputs.commandWorkPos := FALSE;
   instcmStackTableVaccum.statCurrentInputs.reset := FALSE;
   instcmStackTableVaccum.statPreviousInputs.commandHomePos := FALSE;
   instcmStackTableVaccum.statPreviousInputs.commandWorkPos := FALSE;
   instcmStackTableVaccum.statPreviousInputs.reset := FALSE;
   instcmStackTableVaccum.statCurrentInterface.commandHomePos := FALSE;
   instcmStackTableVaccum.statCurrentInterface.commandWorkPos := FALSE;
   instcmStackTableVaccum.statCurrentInterface.reset := FALSE;
   instcmStackTableVaccum.statPreviousInterface.commandHomePos := FALSE;
   instcmStackTableVaccum.statPreviousInterface.commandWorkPos := FALSE;
   instcmStackTableVaccum.statPreviousInterface.reset := FALSE;
   instcmStackTableVaccum.statEmptyDiagnostics.status := 16#0000;
   instcmStackTableVaccum.statEmptyDiagnostics.subfunctionStatus := 16#0000;
   instcmStackTableVaccum.statEmptyDiagnostics.stateNumber := 0;
   instcmStackTableVaccum.instTimerReachPos.PT := T#0MS;
   instcmStackTableVaccum.instTimerReachPos.IN := FALSE;
   instcmStackTableVaccum.instTimerLeavePos.PT := T#0MS;
   instcmStackTableVaccum.instTimerLeavePos.IN := FALSE;
   instcmStackTableVaccum.instTimerDiscrepancyCheck.PT := T#0MS;
   instcmStackTableVaccum.instTimerDiscrepancyCheck.IN := FALSE;
   instcmStackTableVaccum.statDisableAlarms := FALSE;
   instcmStackTableVaccum.statDiagnostics.status := 16#7003;
   instcmStackTableVaccum.statDiagnostics.subfunctionStatus := 16#0000;
   instcmStackTableVaccum.statDiagnostics.stateNumber := 0;
   instcmStackTableVaccum.statEnablePrevious := TRUE;
   instcmStackTableVaccum.statFirstCall := FALSE;
   instcmStackTableVaccum.statResetPrevious := FALSE;
   instcmStackTableVaccum.statValid := TRUE;
   instcmStackTableVaccum.statBusy := TRUE;
   instcmStackTableVaccum.statError := FALSE;
   instcmStackTableVaccum.statInterlockWorkOff := FALSE;
   instcmStackTableVaccum.statInterlockHomeOff := FALSE;
   instcmStackTableVaccum.statFbState := 50;
   instcmStackTableVaccum.statFbStatePrevious := 50;
   instcmStackTableVaccum.statErrorUserCleared := FALSE;
   instcmStackTableVaccum.statErrorAutoCleared := FALSE;
   instcmStackTableVaccum.statErrorState := 16#0000;
   instcmStackTableVaccum.statDisablingCompleted := FALSE;
   instcmStackTableVaccum.statFeedbackHomePos := TRUE;
   instcmStackTableVaccum.statFeedbackWorkPos := FALSE;
   instcmStackTableGapPadUpDown.enable := TRUE;
   instcmStackTableGapPadUpDown.parentReferenceDesignator := WSTRING#'';
   instcmStackTableGapPadUpDown.feedbackHomePos := TRUE;
   instcmStackTableGapPadUpDown.feedbackWorkPos := FALSE;
   instcmStackTableGapPadUpDown.enableManualCmds := TRUE;
   instcmStackTableGapPadUpDown.interlockWorkPos := TRUE;
   instcmStackTableGapPadUpDown.interlockHomePos := TRUE;
   instcmStackTableGapPadUpDown.goToHomePos := FALSE;
   instcmStackTableGapPadUpDown.goToWorkPos := FALSE;
   instcmStackTableGapPadUpDown.statProcessValues.enable := TRUE;
   instcmStackTableGapPadUpDown.statProcessValues.referenceDesignator := WSTRING#'StackTableGapPadUpDown';
   instcmStackTableGapPadUpDown.statProcessValues.commandHomePos := FALSE;
   instcmStackTableGapPadUpDown.statProcessValues.commandWorkPos := FALSE;
   instcmStackTableGapPadUpDown.statProcessValues.goToHomePos := FALSE;
   instcmStackTableGapPadUpDown.statProcessValues.goToWorkPos := FALSE;
   instcmStackTableGapPadUpDown.statProcessValues.inHomePos := FALSE;
   instcmStackTableGapPadUpDown.statProcessValues.inWorkPos := FALSE;
   instcmStackTableGapPadUpDown.statProcessValues.reset := FALSE;
   instcmStackTableGapPadUpDown.statProcessValues.enableManualCmds := TRUE;
   instcmStackTableGapPadUpDown.statProcessValues.error := FALSE;
   instcmStackTableGapPadUpDown.statProcessValues.interlockHomePos := TRUE;
   instcmStackTableGapPadUpDown.statProcessValues.interlockWorkPos := TRUE;
   instcmStackTableGapPadUpDown.statProcessValues.status := 16#7003;
   instcmStackTableGapPadUpDown.statProcessValues.interlockWarningWorkPos := FALSE;
   instcmStackTableGapPadUpDown.statProcessValues.interlockWarningHomePos := FALSE;
   instcmStackTableGapPadUpDown.statCurrentInputs.commandHomePos := FALSE;
   instcmStackTableGapPadUpDown.statCurrentInputs.commandWorkPos := FALSE;
   instcmStackTableGapPadUpDown.statCurrentInputs.reset := FALSE;
   instcmStackTableGapPadUpDown.statPreviousInputs.commandHomePos := FALSE;
   instcmStackTableGapPadUpDown.statPreviousInputs.commandWorkPos := FALSE;
   instcmStackTableGapPadUpDown.statPreviousInputs.reset := FALSE;
   instcmStackTableGapPadUpDown.statCurrentInterface.commandHomePos := FALSE;
   instcmStackTableGapPadUpDown.statCurrentInterface.commandWorkPos := FALSE;
   instcmStackTableGapPadUpDown.statCurrentInterface.reset := FALSE;
   instcmStackTableGapPadUpDown.statPreviousInterface.commandHomePos := FALSE;
   instcmStackTableGapPadUpDown.statPreviousInterface.commandWorkPos := FALSE;
   instcmStackTableGapPadUpDown.statPreviousInterface.reset := FALSE;
   instcmStackTableGapPadUpDown.statEmptyDiagnostics.status := 16#0000;
   instcmStackTableGapPadUpDown.statEmptyDiagnostics.subfunctionStatus := 16#0000;
   instcmStackTableGapPadUpDown.statEmptyDiagnostics.stateNumber := 0;
   instcmStackTableGapPadUpDown.instTimerReachPos.PT := T#0MS;
   instcmStackTableGapPadUpDown.instTimerReachPos.IN := FALSE;
   instcmStackTableGapPadUpDown.instTimerLeavePos.PT := T#0MS;
   instcmStackTableGapPadUpDown.instTimerLeavePos.IN := FALSE;
   instcmStackTableGapPadUpDown.instTimerDiscrepancyCheck.PT := T#0MS;
   instcmStackTableGapPadUpDown.instTimerDiscrepancyCheck.IN := FALSE;
   instcmStackTableGapPadUpDown.statDisableAlarms := FALSE;
   instcmStackTableGapPadUpDown.statDiagnostics.status := 16#7003;
   instcmStackTableGapPadUpDown.statDiagnostics.subfunctionStatus := 16#0000;
   instcmStackTableGapPadUpDown.statDiagnostics.stateNumber := 0;
   instcmStackTableGapPadUpDown.statEnablePrevious := TRUE;
   instcmStackTableGapPadUpDown.statFirstCall := FALSE;
   instcmStackTableGapPadUpDown.statResetPrevious := FALSE;
   instcmStackTableGapPadUpDown.statValid := TRUE;
   instcmStackTableGapPadUpDown.statBusy := TRUE;
   instcmStackTableGapPadUpDown.statError := FALSE;
   instcmStackTableGapPadUpDown.statInterlockWorkOff := FALSE;
   instcmStackTableGapPadUpDown.statInterlockHomeOff := FALSE;
   instcmStackTableGapPadUpDown.statFbState := 50;
   instcmStackTableGapPadUpDown.statFbStatePrevious := 50;
   instcmStackTableGapPadUpDown.statErrorUserCleared := FALSE;
   instcmStackTableGapPadUpDown.statErrorAutoCleared := FALSE;
   instcmStackTableGapPadUpDown.statErrorState := 16#0000;
   instcmStackTableGapPadUpDown.statDisablingCompleted := FALSE;
   instcmStackTableGapPadUpDown.statFeedbackHomePos := TRUE;
   instcmStackTableGapPadUpDown.statFeedbackWorkPos := FALSE;
   instManageAlarms.proDiagState.Total_Number := 492;
   instManageAlarms.proDiagState.All := TRUE;
   instManageAlarms.proDiagState.O := FALSE;
   instManageAlarms.proDiagState.I := FALSE;
   instManageAlarms.proDiagState.R := FALSE;
   instManageAlarms.proDiagState."A" := FALSE;
   instManageAlarms.proDiagState.P := FALSE;
   instManageAlarms.proDiagState.Merr := TRUE;
   instManageAlarms.proDiagState.Mtxt := FALSE;
   instManageAlarms.proDiagState.SV_Types := 16#20;
   instManageAlarms.proDiagState.C1 := TRUE;
   instManageAlarms.proDiagState.C2 := FALSE;
   instManageAlarms.proDiagState.C3 := FALSE;
   instManageAlarms.proDiagState.C4 := FALSE;
   instManageAlarms.proDiagState.C5 := FALSE;
   instManageAlarms.proDiagState.C6 := FALSE;
   instManageAlarms.proDiagState.C7 := FALSE;
   instManageAlarms.proDiagState.C8 := FALSE;
   instManageAlarms.proDiagState.Categories := 16#01;
   instManageAlarms.proDiagState.Sub_Cat_1 := 16#0000_0001;
   instManageAlarms.proDiagState.Sub_Cat_2 := 16#0000_0000;
   instManageAlarms.proDiagState.Reserved := 16#00;
   instManageAlarms.parentAlarmDB.error := TRUE;
   instManageAlarms.parentAlarmDB.warning := FALSE;
   instManageAlarms.parentAlarmDB.info := FALSE;
   instManageAlarms.alarmDB.error := TRUE;
   instManageAlarms.alarmDB.warning := FALSE;
   instManageAlarms.alarmDB.info := FALSE;
   instManageAlarms.hmiInterfaceDB.error := TRUE;
   instManageAlarms.hmiInterfaceDB.warning := FALSE;
   instManageAlarms.hmiInterfaceDB.info := FALSE;
   statUnitStatus.acknowledgeActive := FALSE;
   statUnitStatus.alarmsDisabled := FALSE;
   statUnitStatus.simulationActive := FALSE;
   statUnitStatus.safetyReleased := TRUE;
   statUnitStatus.specialFunctions.GaugeRnR1AnodeAlign := FALSE;
   statUnitStatus.specialFunctions.GaugeRnR1CathodeAlign := FALSE;
   statUnitStatus.specialFunctions.GaugeRnR3AnodeAlign := FALSE;
   statUnitStatus.specialFunctions.GaugeRnR3CathodeAlign := FALSE;
   statUnitStatus.specialFunctions.releaseEntry := FALSE;
   statUnitStatus.specialFunctions.dryRun := FALSE;
   statUnitStatus.specialFunctions.ReelCutAnodeUnuse := FALSE;
   statUnitStatus.mode.current := 2;
   statUnitStatus.mode.production := FALSE;
   statUnitStatus.mode.maintenance := TRUE;
   statUnitStatus.mode.manual := FALSE;
   statUnitStatus.mode.sleep := FALSE;
   statUnitStatus.mode.deepsleep := FALSE;
   statUnitStatus.mode.userMode04 := FALSE;
   statUnitStatus.mode.userMode05 := FALSE;
   statUnitStatus.mode.userMode06 := FALSE;
   statUnitStatus.mode.userMode07 := FALSE;
   statUnitStatus.mode.userMode08 := FALSE;
   statUnitStatus.mode.userMode09 := FALSE;
   statUnitStatus.mode.userMode10 := FALSE;
   statUnitStatus.mode.userMode11 := FALSE;
   statUnitStatus.mode.userMode12 := FALSE;
   statUnitStatus.mode.userMode13 := FALSE;
   statUnitStatus.state.current := 2;
   statUnitStatus.state.clearing := FALSE;
   statUnitStatus.state.stopped := TRUE;
   statUnitStatus.state.starting := FALSE;
   statUnitStatus.state.idle := FALSE;
   statUnitStatus.state.suspended := FALSE;
   statUnitStatus.state.execute := FALSE;
   statUnitStatus.state.stopping := FALSE;
   statUnitStatus.state.aborting := FALSE;
   statUnitStatus.state.aborted := FALSE;
   statUnitStatus.state.holding := FALSE;
   statUnitStatus.state.held := FALSE;
   statUnitStatus.state.unholding := FALSE;
   statUnitStatus.state.suspending := FALSE;
   statUnitStatus.state.unsuspending := FALSE;
   statUnitStatus.state.resetting := FALSE;
   statUnitStatus.state.completing := FALSE;
   statUnitStatus.state.complete := FALSE;
END_DATA_BLOCK
